(* Logix 5000 project; controller Hose_HP_Test_Rig_V1 vendor 1 type 14 code 149 rev 32.11; software revision 32.00; part 9 of 10 *)
(* tags used below, declared in another part *)
   ALIGN : SCP;
   CYCLE_TIMER_STN2 : TIMER;
   CYCLE_TIMER_STN3 : TIMER;
   GOTO_FAIL_BIN_STN1 : DINT;
   GOTO_FAULT_BIN_STN3 : DINT;
   GOTO_FAULT_BIN_STN4 : DINT;
   INDV_LTEST_ON_STN1 : BOOL;
   INDV_LTEST_ON_STN2 : BOOL;
   INDV_LTEST_ON_STN3 : BOOL;
   ONS1 : BOOL;
   ONS10 : BOOL;
   ONS11 : BOOL;
   ONS12 : BOOL;
   ONS13 : BOOL;
   ONS14 : BOOL;
   ONS15 : BOOL;
   ONS16 : BOOL;
   ONS17 : BOOL;
   ONS18 : BOOL;
   ONS19 : BOOL;
   ONS2 : BOOL;
   ONS20 : BOOL;
   ONS21 : BOOL;
   ONS22 : BOOL;
   ONS23 : BOOL;
   ONS24 : BOOL;
   ONS25 : BOOL;
   ONS3 : BOOL;
   ONS54 : BOOL;
   ONS55 : BOOL;
   ONS56 : BOOL;
   ONS57 : BOOL;
   ONS58 : BOOL;
   ONS59 : BOOL;
   ONS6 : BOOL;
   ONS60 : BOOL;
   ONS61 : BOOL;
   ONS62 : BOOL;
   ONS67 : BOOL;
   ONS68 : BOOL;
   ONS7 : BOOL;
   ONS8 : BOOL;
   ONS9 : BOOL;
   TEST_INIT_DEL_STN2 : TIMER;
   TEST_INIT_DEL_STN3 : TIMER;
   TIME1 : TIMER;
   ACT_DROP_STN1 : REAL;
   ACT_DROP_STN2 : REAL;
   ACT_DROP_STN3 : REAL;
   ACT_DROP_STN4 : REAL;
   ACT_PR_STN1 : REAL;
   ACT_PR_STN2 : REAL;
   ACT_PR_STN3 : REAL;
   ACT_PR_STN4 : REAL;
   ACT_TRAVEL : REAL;
   AUTO_DOOR_OPEN_SEQ : DINT;
   AUTO_DOOR_OPEN_SEQ_STN2 : DINT;
   AUTO_DOOR_OPEN_SEQ_STN3 : DINT;
   AUTO_TEST_ON_STN1 : BOOL;
   AUTO_TEST_ON_STN2 : BOOL;
   AUTO_TEST_ON_STN3 : BOOL;
   AUTO_TEST_ON_STN4 : BOOL;
   AUTO_TEST_OVER_STN1 : BOOL;
   AUTO_TEST_OVER_STN2 : BOOL;
   AUTO_TEST_OVER_STN3 : BOOL;
   AUTO_TEST_OVER_STN4 : BOOL;
   AUTO_TEST_SEL_STN1 : BOOL;
   AUTO_TEST_SEL_STN2 : BOOL;
   AUTO_TEST_SEL_STN3 : BOOL;
   AUTO_TEST_SEL_STN4 : BOOL;
   BOTTOM_CLAMP_PS_STN1 : ALIAS FOR Local:1:I.Data.13;
   BOTTOM_CLAMP_PS_STN2 : ALIAS FOR Local:2:I.Data.2;
   BOTTOM_CLAMP_PS_STN3 : ALIAS FOR Local:2:I.Data.7;
   BOTTOM_CLAMP_PS_STN4 : ALIAS FOR Local:2:I.Data.12;
   BOTTOM_CLAMP_SEL_STN1 : BOOL;
   BOTTOM_CLAMP_SEL_STN2 : BOOL;
   BOTTOM_CLAMP_SEL_STN3 : BOOL;
   BOTTOM_CLAMP_SEL_STN4 : BOOL;
   BOTTOM_CLAMP_SEQ_STN1 : DINT;
   BOTTOM_CLAMP_SEQ_STN2 : DINT;
   BOTTOM_CLAMP_SEQ_STN3 : DINT;
   BOTTOM_CLAMP_SET_STN1 : BOOL;
   BOTTOM_CLAMP_SET_STN2 : BOOL;
   BOTTOM_CLAMP_SET_STN3 : BOOL;
   BOTTOM_CLAMP_SET_STN4 : BOOL;
   BOTTOM_DECLAMP_SEQ_STN2 : DINT;
   BOTTOM_DECLAMP_SEQ_STN3 : DINT;
   BOTTOM_DECLAMP_SET_STN1 : BOOL;
   BOTTOM_DECLAMP_SET_STN2 : BOOL;
   BOTTOM_DECLAMP_SET_STN3 : BOOL;
   BOTTOM_DECLAMP_SET_STN4 : BOOL;
   CLR_ONS_STN1 : BOOL;
   CLR_ONS_STN2 : BOOL;
   CLR_ONS_STN3 : BOOL;
   CONS_CALB_OFF_STN1 : BOOL;
   CONS_CALB_OFF_STN2 : BOOL;
   CONS_CALB_OFF_STN3 : BOOL;
   CONS_CALB_OFF_STN4 : BOOL;
   CONS_CALB_ON_STN1 : BOOL;
   CONS_CALB_ON_STN2 : BOOL;
   CONS_CALB_ON_STN3 : BOOL;
   CONS_CALB_ON_STN4 : BOOL;
   CONS_RESULT_STN1 : DINT;
   CONS_RESULT_STN2 : DINT;
   CONS_RESULT_STN3 : DINT;
   CONS_RESULT_STN4 : DINT;
   CONS_STS_STN1 : DINT;
   CONS_STS_STN2 : DINT;
   CONS_STS_STN3 : DINT;
   CONS_STS_STN4 : DINT;
   CONS_TEST_ON : BOOL;
   CONSTRICTION_CALB_SEL_STN1 : BOOL;
   CONSTRICTION_CALB_SEL_STN2 : BOOL;
   CONSTRICTION_CALB_SEL_STN3 : BOOL;
   CONSTRICTION_CALB_SEL_STN4 : BOOL;
   CONSTRICTION_VALVE_STN1 : BOOL;
   CONSTRICTION_VALVE_STN2 : BOOL;
   CONSTRICTION_VALVE_STN3 : BOOL;
   CONSTRICTION_VALVE_STN4 : BOOL;
   CRIMP_PASS : ALIAS FOR Local:2:I.Data.31;
   CRIMP_PASS_TO_TRACE : DINT;
   CYCLE_START_PB_STN1 : ALIAS FOR Local:1:I.Data.2;
   CYCLE_TIME_ACT_STN1 : REAL;
   CYCLE_TIME_ACT_STN2 : REAL;
   CYCLE_TIME_ACT_STN3 : REAL;
   CYCLE_TIME_ACT_STN4 : REAL;
   CYCLE_TIMER_STN1 : TIMER;
   CYCLE_TIMER_STN4 : TIMER;
   DOOR_CLAMP_SET_STN1 : SETTING_MODE;
   DOOR_CLAMP_SET_STN2 : SETTING_MODE;
   DOOR_CLAMP_SET_STN3 : SETTING_MODE;
   DOOR_CLAMP_SET_STN4 : SETTING_MODE;
   DOOR_CLOSE_SEL_STN1 : BOOL;
   DOOR_CLOSE_SEL_STN2 : BOOL;
   DOOR_CLOSE_SEL_STN3 : BOOL;
   DOOR_CLOSE_SEL_STN4 : BOOL;
   DOOR_CLOSE_SET_STN1 : BOOL;
   DOOR_CLOSE_SET_STN2 : BOOL;
   DOOR_CLOSE_SET_STN3 : BOOL;
   DOOR_CLOSE_SET_STN4 : BOOL;
   DOOR_OPEN_RS_STN1 : ALIAS FOR Local:1:I.Data.10;
   DOOR_OPEN_RS_STN2 : ALIAS FOR Local:1:I.Data.15;
   DOOR_OPEN_RS_STN3 : ALIAS FOR Local:2:I.Data.4;
   DOOR_OPEN_RS_STN4 : ALIAS FOR Local:2:I.Data.10;
   DOOR_OPEN_SET_STN1 : BOOL;
   DOOR_OPEN_SET_STN2 : BOOL;
   DOOR_OPEN_SET_STN3 : BOOL;
   DOOR_OPEN_SET_STN4 : BOOL;
   EXHAUST_SET_STN1 : BOOL;
   EXHAUST_SET_STN2 : BOOL;
   EXHAUST_SET_STN3 : BOOL;
   EXHAUST_SET_STN4 : BOOL;
   EXHAUST_VALVE_STN1 : ALIAS FOR Local:1:O.Data.7;
   EXHAUST_VALVE_STN2 : ALIAS FOR Local:1:O.Data.15;
   EXHAUST_VALVE_STN3 : ALIAS FOR Local:3:O.Data.7;
   EXHAUST_VALVE_STN4 : ALIAS FOR Local:3:O.Data.15;
   FAIL_BIN_DOOR_PROXY : ALIAS FOR Local:2:I.Data.29;
   FAILED_STN1 : BOOL;
   FAILED_STN2 : BOOL;
   FAILED_STN3 : BOOL;
   FAILED_STN4 : BOOL;
   FAULTED_STN1 : BOOL;
   FAULTED_STN2 : BOOL;
   FAULTED_STN3 : BOOL;
   FAULTED_STN4 : BOOL;
   FIX_DOWN_SET : BOOL;
   FIX_UP_SET : BOOL;
   GOTO_FAIL_BIN_STN2 : DINT;
   GOTO_FAIL_BIN_STN3 : DINT;
   GOTO_FAIL_BIN_STN4 : DINT;
   GOTO_FAULT_BIN_STN1 : DINT;
   GOTO_FAULT_BIN_STN2 : DINT;
   HOME_COND_OK_STN1 : BOOL;
   HOME_COND_OK_STN2 : BOOL;
   HOME_COND_OK_STN3 : BOOL;
   HOME_COND_OK_STN4 : BOOL;
   HP_ACT_DROP_STN1 : REAL;
   HP_ACT_DROP_STN2 : REAL;
   HP_ACT_DROP_STN3 : REAL;
   HP_ACT_DROP_STN4 : REAL;
   HP_ACT_PR_STN1 : REAL;
   HP_ACT_PR_STN2 : REAL;
   HP_ACT_PR_STN3 : REAL;
   HP_ACT_PR_STN4 : REAL;
   HP_RESULT_STN1 : DINT;
   HP_RESULT_STN2 : DINT;
   HP_RESULT_STN3 : DINT;
   HP_RESULT_STN4 : DINT;
   HP_SENSOR_SEL : BOOL;
   HP_STS_STN1 : DINT;
   HP_STS_STN2 : DINT;
   HP_STS_STN3 : DINT;
   HP_STS_STN4 : DINT;
   HP_TEST_ON : BOOL;
   INDV_CTEST_ON_STN1 : BOOL;
   INDV_CTEST_ON_STN2 : BOOL;
   INDV_CTEST_ON_STN3 : BOOL;
   INIT_STN1 : BOOL;
   INIT_STN2 : BOOL;
   INIT_STN3 : BOOL;
   LH_START_PB_STN2 : ALIAS FOR Local:1:I.Data.3;
   LH_START_PB_STN3 : ALIAS FOR Local:1:I.Data.4;
   LH_START_PB_STN4 : ALIAS FOR Local:1:I.Data.5;
   LOGIN_LEVEL : INT;
   MASTER_WORK_MAIN_MENU_EN : BOOL;
   MOTOR_DOWN : ALIAS FOR REM:O.Data[1].3;
   MOTOR_SAFETY : BOOL;
   MOTOR_UP : ALIAS FOR REM:O.Data[1].2;
   MSG_STN1 : DINT;
   MSG_STN2 : DINT;
   MSG_STN3 : DINT;
   MSG_STN4 : DINT;
   ONS5 : BOOL;
   OTHER_CAL_EDIT_MODE : BOOL;
   OTHER_CAL_VIEW_MODE : BOOL;
   OTHER_SENSOR_SEL : BOOL;
   PASSED_STN1 : BOOL;
   PASSED_STN2 : BOOL;
   PASSED_STN3 : BOOL;
   RETEST : BOOL;
   RST_SEQ_ON_STN1 : BOOL;
   RST_SEQ_ON_STN2 : BOOL;
   RST_SEQ_ON_STN3 : BOOL;
   RST_SEQ_ON_STN4 : BOOL;
   SCR_STS : DINT[6];
   SENS_CAL_EDIT_MODE : BOOL;
   SENS_CAL_SEL_BOTTOM_CLAMP : BOOL;
   SENS_CAL_SEL_MASTER : BOOL;
   SENS_CAL_SEL_STAMP : BOOL;
   SENS_CAL_SEL_TOP_CLAMP : BOOL;
   SENS_CAL_VIEW_MODE : BOOL;
   SENS_CALB_SEL_STN1 : BOOL;
   SENS_CALB_SEL_STN2 : BOOL;
   SENS_CALB_SEL_STN3 : BOOL;
   SENS_CALB_SEL_STN4 : BOOL;
   SEQ_NO_STN1 : DINT;
   SEQ_NO_STN2 : DINT;
   SEQ_NO_STN3 : DINT;
   SET_240 : REAL;
   SET_DISTANCE : REAL;
   SET_MENU_STN1_EN : BOOL;
   SET_MENU_STN2_EN : BOOL;
   SET_MENU_STN3_EN : BOOL;
   SET_MENU_STN4_EN : BOOL;
   SET_MODE_SEL_STN1 : BOOL;
   SET_MODE_SEL_STN2 : BOOL;
   SET_MODE_SEL_STN3 : BOOL;
   SET_MODE_SEL_STN4 : BOOL;
   SET_TIMER : REAL;
   SLIDE_TRAVEL : TIMER;
(* MainProgram, continued *)

ROUTINE SENS_CALB   (* ladder *)
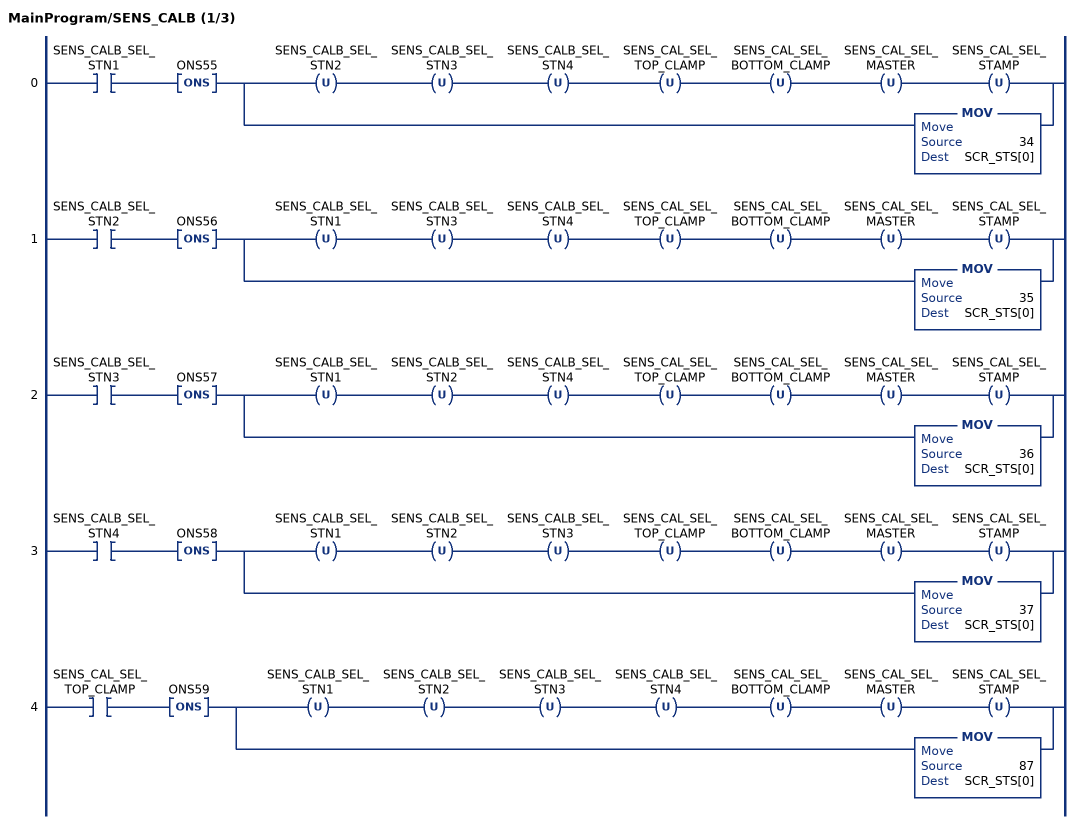
   0: XIC(SENS_CALB_SEL_STN1)ONS(ONS55)[OTU(SENS_CALB_SEL_STN2) OTU(SENS_CALB_SEL_STN3) OTU(SENS_CALB_SEL_STN4) OTU(SENS_CAL_SEL_TOP_CLAMP) OTU(SENS_CAL_SEL_BOTTOM_CLAMP) OTU(SENS_CAL_SEL_MASTER) OTU(SENS_CAL_SEL_STAMP) ,MOV(34,SCR_STS[0]) ];
   1: XIC(SENS_CALB_SEL_STN2)ONS(ONS56)[OTU(SENS_CALB_SEL_STN1) OTU(SENS_CALB_SEL_STN3) OTU(SENS_CALB_SEL_STN4) OTU(SENS_CAL_SEL_TOP_CLAMP) OTU(SENS_CAL_SEL_BOTTOM_CLAMP) OTU(SENS_CAL_SEL_MASTER) OTU(SENS_CAL_SEL_STAMP) ,MOV(35,SCR_STS[0]) ];
   2: XIC(SENS_CALB_SEL_STN3)ONS(ONS57)[OTU(SENS_CALB_SEL_STN1) OTU(SENS_CALB_SEL_STN2) OTU(SENS_CALB_SEL_STN4) OTU(SENS_CAL_SEL_TOP_CLAMP) OTU(SENS_CAL_SEL_BOTTOM_CLAMP) OTU(SENS_CAL_SEL_MASTER) OTU(SENS_CAL_SEL_STAMP) ,MOV(36,SCR_STS[0]) ];
   3: XIC(SENS_CALB_SEL_STN4)ONS(ONS58)[OTU(SENS_CALB_SEL_STN1) OTU(SENS_CALB_SEL_STN2) OTU(SENS_CALB_SEL_STN3) OTU(SENS_CAL_SEL_TOP_CLAMP) OTU(SENS_CAL_SEL_BOTTOM_CLAMP) OTU(SENS_CAL_SEL_MASTER) OTU(SENS_CAL_SEL_STAMP) ,MOV(37,SCR_STS[0]) ];
   4: XIC(SENS_CAL_SEL_TOP_CLAMP)ONS(ONS59)[OTU(SENS_CALB_SEL_STN1) OTU(SENS_CALB_SEL_STN2) OTU(SENS_CALB_SEL_STN3) OTU(SENS_CALB_SEL_STN4) OTU(SENS_CAL_SEL_BOTTOM_CLAMP) OTU(SENS_CAL_SEL_MASTER) OTU(SENS_CAL_SEL_STAMP) ,MOV(87,SCR_STS[0]) ];
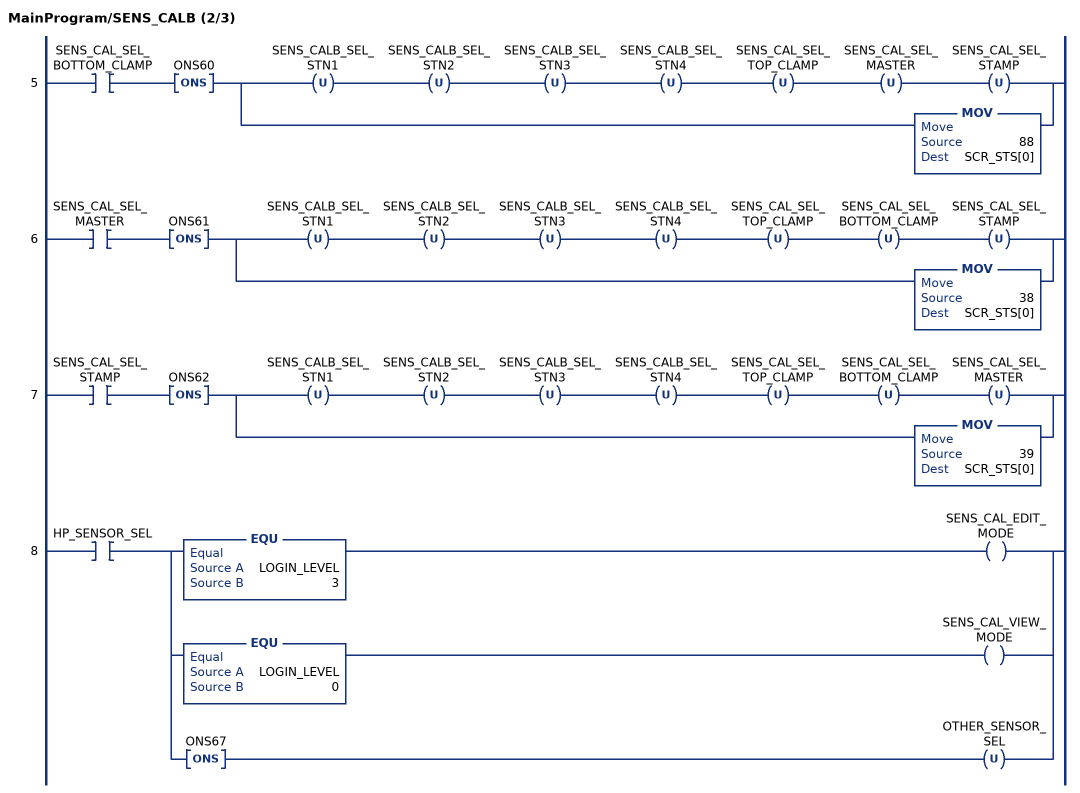
   5: XIC(SENS_CAL_SEL_BOTTOM_CLAMP)ONS(ONS60)[OTU(SENS_CALB_SEL_STN1) OTU(SENS_CALB_SEL_STN2) OTU(SENS_CALB_SEL_STN3) OTU(SENS_CALB_SEL_STN4) OTU(SENS_CAL_SEL_TOP_CLAMP) OTU(SENS_CAL_SEL_MASTER) OTU(SENS_CAL_SEL_STAMP) ,MOV(88,SCR_STS[0]) ];
   6: XIC(SENS_CAL_SEL_MASTER)ONS(ONS61)[OTU(SENS_CALB_SEL_STN1) OTU(SENS_CALB_SEL_STN2) OTU(SENS_CALB_SEL_STN3) OTU(SENS_CALB_SEL_STN4) OTU(SENS_CAL_SEL_TOP_CLAMP) OTU(SENS_CAL_SEL_BOTTOM_CLAMP) OTU(SENS_CAL_SEL_STAMP) ,MOV(38,SCR_STS[0]) ];
   7: XIC(SENS_CAL_SEL_STAMP)ONS(ONS62)[OTU(SENS_CALB_SEL_STN1) OTU(SENS_CALB_SEL_STN2) OTU(SENS_CALB_SEL_STN3) OTU(SENS_CALB_SEL_STN4) OTU(SENS_CAL_SEL_TOP_CLAMP) OTU(SENS_CAL_SEL_BOTTOM_CLAMP) OTU(SENS_CAL_SEL_MASTER) ,MOV(39,SCR_STS[0]) ];
   8: XIC(HP_SENSOR_SEL)[EQU(LOGIN_LEVEL,3) OTE(SENS_CAL_EDIT_MODE) ,EQU(LOGIN_LEVEL,0) OTE(SENS_CAL_VIEW_MODE) ,ONS(ONS67) OTU(OTHER_SENSOR_SEL) ];
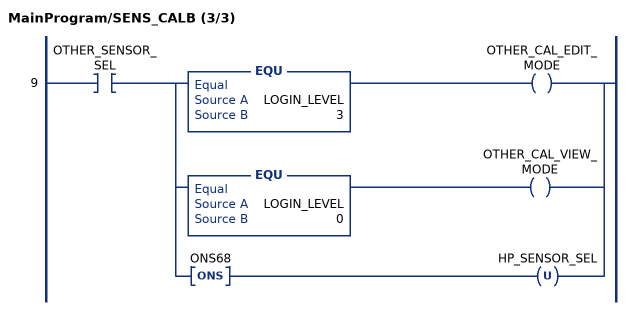
   9: XIC(OTHER_SENSOR_SEL)[EQU(LOGIN_LEVEL,3) OTE(OTHER_CAL_EDIT_MODE) ,EQU(LOGIN_LEVEL,0) OTE(OTHER_CAL_VIEW_MODE) ,ONS(ONS68) OTU(HP_SENSOR_SEL) ];
END_ROUTINE

ROUTINE Setting_Mode   (* ladder *)
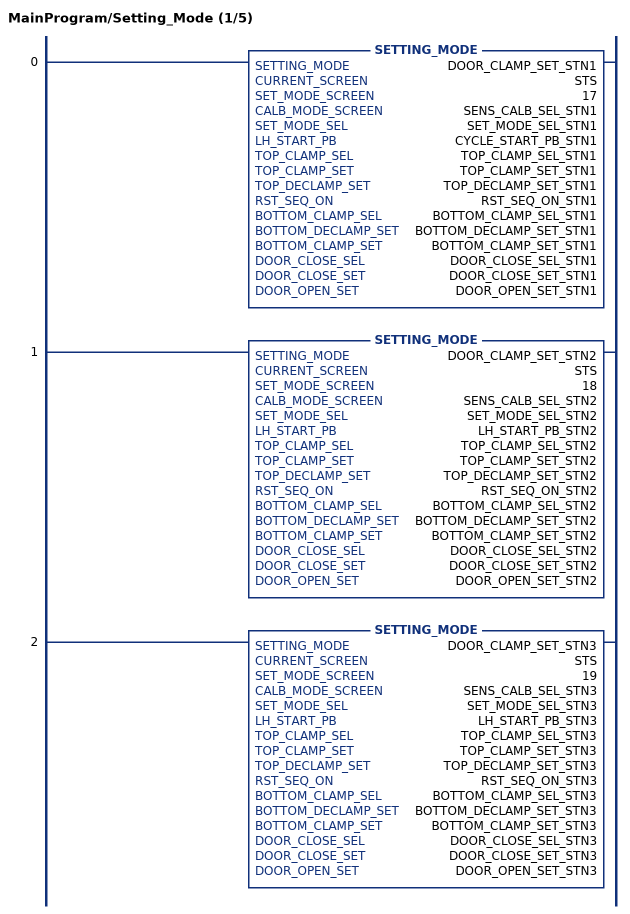
   0: SETTING_MODE(DOOR_CLAMP_SET_STN1,STS,17,SENS_CALB_SEL_STN1,SET_MODE_SEL_STN1,CYCLE_START_PB_STN1,TOP_CLAMP_SEL_STN1,TOP_CLAMP_SET_STN1,TOP_DECLAMP_SET_STN1,RST_SEQ_ON_STN1,BOTTOM_CLAMP_SEL_STN1,BOTTOM_DECLAMP_SET_STN1,BOTTOM_CLAMP_SET_STN1,DOOR_CLOSE_SEL_STN1,DOOR_CLOSE_SET_STN1,DOOR_OPEN_SET_STN1);
   1: SETTING_MODE(DOOR_CLAMP_SET_STN2,STS,18,SENS_CALB_SEL_STN2,SET_MODE_SEL_STN2,LH_START_PB_STN2,TOP_CLAMP_SEL_STN2,TOP_CLAMP_SET_STN2,TOP_DECLAMP_SET_STN2,RST_SEQ_ON_STN2,BOTTOM_CLAMP_SEL_STN2,BOTTOM_DECLAMP_SET_STN2,BOTTOM_CLAMP_SET_STN2,DOOR_CLOSE_SEL_STN2,DOOR_CLOSE_SET_STN2,DOOR_OPEN_SET_STN2);
   2: SETTING_MODE(DOOR_CLAMP_SET_STN3,STS,19,SENS_CALB_SEL_STN3,SET_MODE_SEL_STN3,LH_START_PB_STN3,TOP_CLAMP_SEL_STN3,TOP_CLAMP_SET_STN3,TOP_DECLAMP_SET_STN3,RST_SEQ_ON_STN3,BOTTOM_CLAMP_SEL_STN3,BOTTOM_DECLAMP_SET_STN3,BOTTOM_CLAMP_SET_STN3,DOOR_CLOSE_SEL_STN3,DOOR_CLOSE_SET_STN3,DOOR_OPEN_SET_STN3);
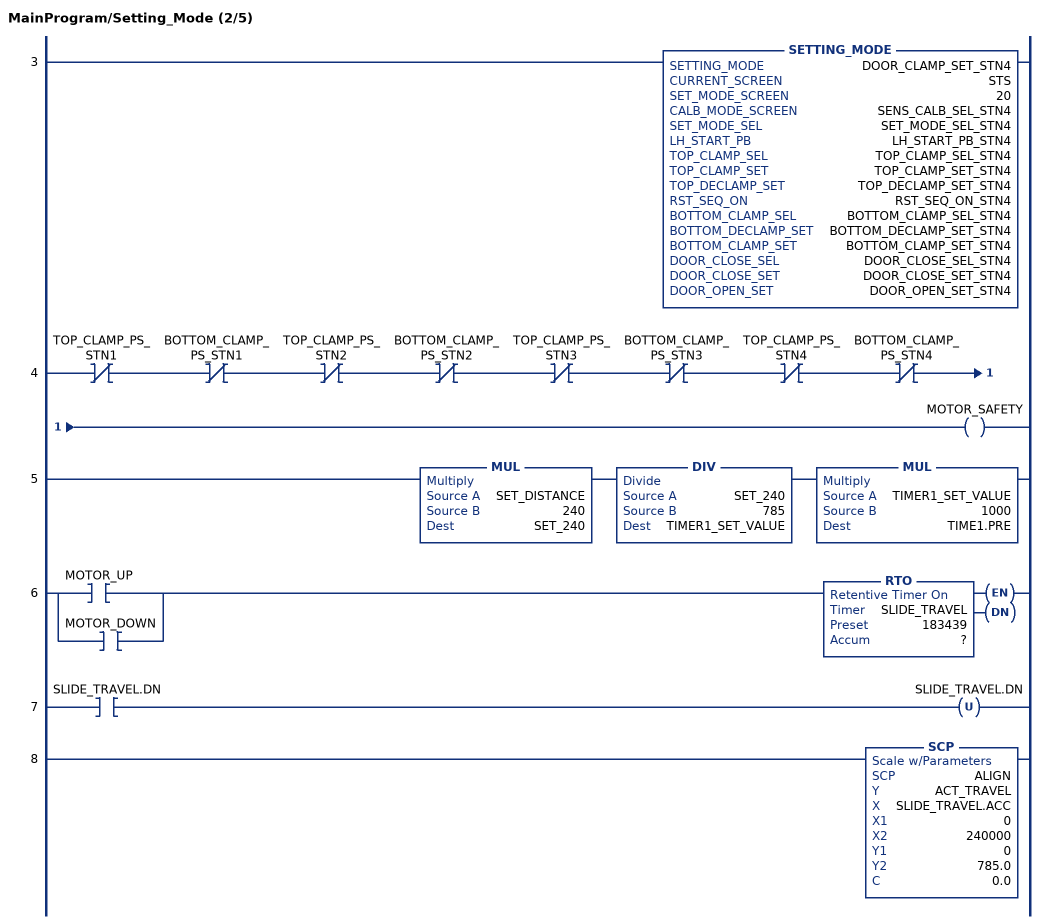
   3: SETTING_MODE(DOOR_CLAMP_SET_STN4,STS,20,SENS_CALB_SEL_STN4,SET_MODE_SEL_STN4,LH_START_PB_STN4,TOP_CLAMP_SEL_STN4,TOP_CLAMP_SET_STN4,TOP_DECLAMP_SET_STN4,RST_SEQ_ON_STN4,BOTTOM_CLAMP_SEL_STN4,BOTTOM_DECLAMP_SET_STN4,BOTTOM_CLAMP_SET_STN4,DOOR_CLOSE_SEL_STN4,DOOR_CLOSE_SET_STN4,DOOR_OPEN_SET_STN4);
   4: XIO(TOP_CLAMP_PS_STN1)XIO(BOTTOM_CLAMP_PS_STN1)XIO(TOP_CLAMP_PS_STN2)XIO(BOTTOM_CLAMP_PS_STN2)XIO(TOP_CLAMP_PS_STN3)XIO(BOTTOM_CLAMP_PS_STN3)XIO(TOP_CLAMP_PS_STN4)XIO(BOTTOM_CLAMP_PS_STN4)OTE(MOTOR_SAFETY);
   5: MUL(SET_DISTANCE,240,SET_240)DIV(SET_240,785,TIMER1_SET_VALUE)MUL(TIMER1_SET_VALUE,1000,TIME1.PRE);
   6: [XIC(MOTOR_UP) ,XIC(MOTOR_DOWN) ]RTO(SLIDE_TRAVEL,?,?);
   7: XIC(SLIDE_TRAVEL.DN)OTU(SLIDE_TRAVEL.DN);
   8: SCP(ALIGN,ACT_TRAVEL,SLIDE_TRAVEL.ACC,0,240000,0,785.0,0.0);
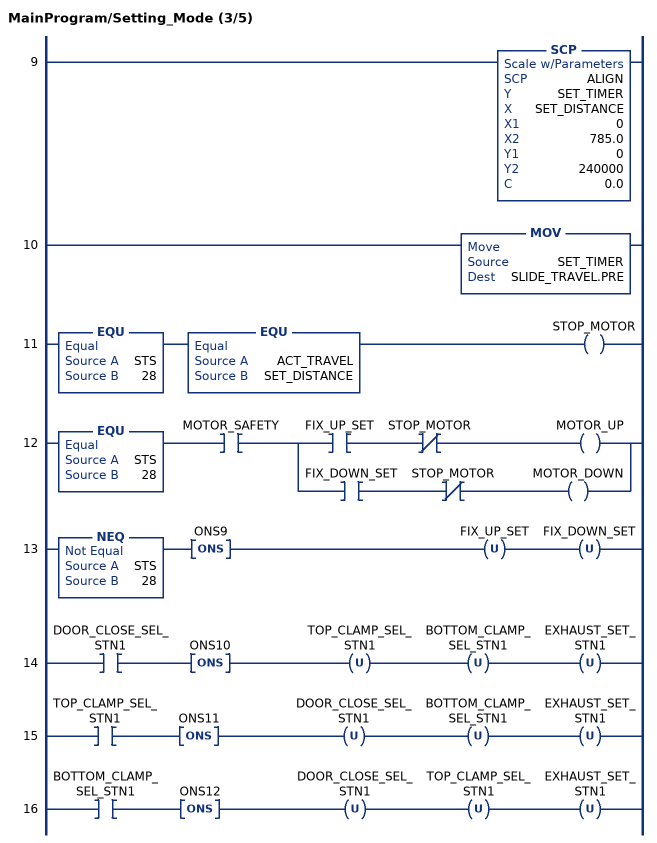
   9: SCP(ALIGN,SET_TIMER,SET_DISTANCE,0,785.0,0,240000,0.0);
   10: MOV(SET_TIMER,SLIDE_TRAVEL.PRE);
   11: EQU(STS,28)EQU(ACT_TRAVEL,SET_DISTANCE)OTE(STOP_MOTOR);
   12: EQU(STS,28)XIC(MOTOR_SAFETY)[XIC(FIX_UP_SET) XIO(STOP_MOTOR) OTE(MOTOR_UP) ,XIC(FIX_DOWN_SET) XIO(STOP_MOTOR) OTE(MOTOR_DOWN) ];
   13: NEQ(STS,28)ONS(ONS9)OTU(FIX_UP_SET)OTU(FIX_DOWN_SET);
   14: XIC(DOOR_CLOSE_SEL_STN1)ONS(ONS10)OTU(TOP_CLAMP_SEL_STN1)OTU(BOTTOM_CLAMP_SEL_STN1)OTU(EXHAUST_SET_STN1);
   15: XIC(TOP_CLAMP_SEL_STN1)ONS(ONS11)OTU(DOOR_CLOSE_SEL_STN1)OTU(BOTTOM_CLAMP_SEL_STN1)OTU(EXHAUST_SET_STN1);
   16: XIC(BOTTOM_CLAMP_SEL_STN1)ONS(ONS12)OTU(DOOR_CLOSE_SEL_STN1)OTU(TOP_CLAMP_SEL_STN1)OTU(EXHAUST_SET_STN1);
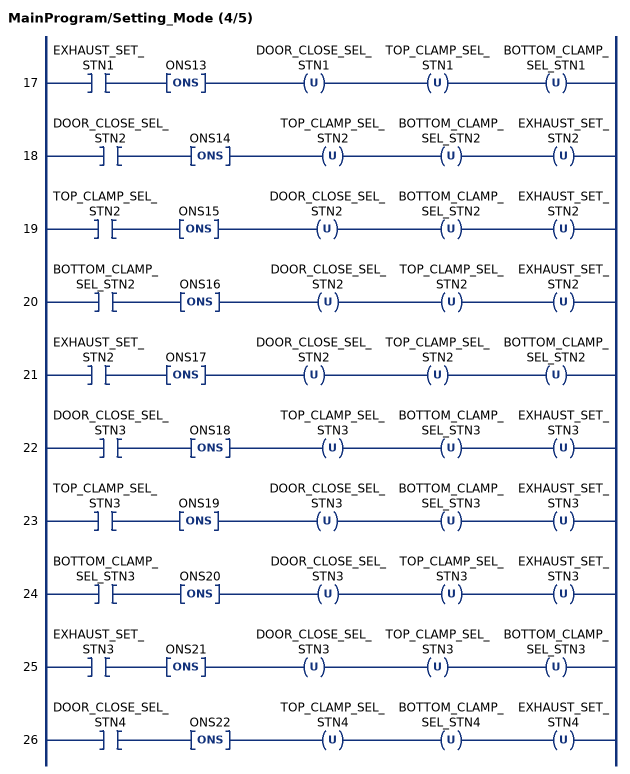
   17: XIC(EXHAUST_SET_STN1)ONS(ONS13)OTU(DOOR_CLOSE_SEL_STN1)OTU(TOP_CLAMP_SEL_STN1)OTU(BOTTOM_CLAMP_SEL_STN1);
   18: XIC(DOOR_CLOSE_SEL_STN2)ONS(ONS14)OTU(TOP_CLAMP_SEL_STN2)OTU(BOTTOM_CLAMP_SEL_STN2)OTU(EXHAUST_SET_STN2);
   19: XIC(TOP_CLAMP_SEL_STN2)ONS(ONS15)OTU(DOOR_CLOSE_SEL_STN2)OTU(BOTTOM_CLAMP_SEL_STN2)OTU(EXHAUST_SET_STN2);
   20: XIC(BOTTOM_CLAMP_SEL_STN2)ONS(ONS16)OTU(DOOR_CLOSE_SEL_STN2)OTU(TOP_CLAMP_SEL_STN2)OTU(EXHAUST_SET_STN2);
   21: XIC(EXHAUST_SET_STN2)ONS(ONS17)OTU(DOOR_CLOSE_SEL_STN2)OTU(TOP_CLAMP_SEL_STN2)OTU(BOTTOM_CLAMP_SEL_STN2);
   22: XIC(DOOR_CLOSE_SEL_STN3)ONS(ONS18)OTU(TOP_CLAMP_SEL_STN3)OTU(BOTTOM_CLAMP_SEL_STN3)OTU(EXHAUST_SET_STN3);
   23: XIC(TOP_CLAMP_SEL_STN3)ONS(ONS19)OTU(DOOR_CLOSE_SEL_STN3)OTU(BOTTOM_CLAMP_SEL_STN3)OTU(EXHAUST_SET_STN3);
   24: XIC(BOTTOM_CLAMP_SEL_STN3)ONS(ONS20)OTU(DOOR_CLOSE_SEL_STN3)OTU(TOP_CLAMP_SEL_STN3)OTU(EXHAUST_SET_STN3);
   25: XIC(EXHAUST_SET_STN3)ONS(ONS21)OTU(DOOR_CLOSE_SEL_STN3)OTU(TOP_CLAMP_SEL_STN3)OTU(BOTTOM_CLAMP_SEL_STN3);
   26: XIC(DOOR_CLOSE_SEL_STN4)ONS(ONS22)OTU(TOP_CLAMP_SEL_STN4)OTU(BOTTOM_CLAMP_SEL_STN4)OTU(EXHAUST_SET_STN4);
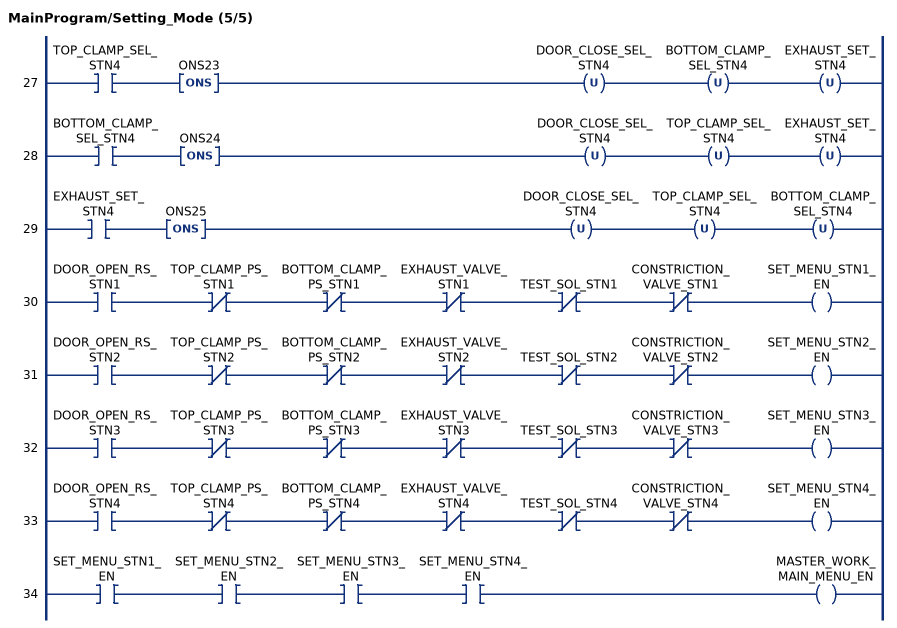
   27: XIC(TOP_CLAMP_SEL_STN4)ONS(ONS23)OTU(DOOR_CLOSE_SEL_STN4)OTU(BOTTOM_CLAMP_SEL_STN4)OTU(EXHAUST_SET_STN4);
   28: XIC(BOTTOM_CLAMP_SEL_STN4)ONS(ONS24)OTU(DOOR_CLOSE_SEL_STN4)OTU(TOP_CLAMP_SEL_STN4)OTU(EXHAUST_SET_STN4);
   29: XIC(EXHAUST_SET_STN4)ONS(ONS25)OTU(DOOR_CLOSE_SEL_STN4)OTU(TOP_CLAMP_SEL_STN4)OTU(BOTTOM_CLAMP_SEL_STN4);
   30: XIC(DOOR_OPEN_RS_STN1)XIO(TOP_CLAMP_PS_STN1)XIO(BOTTOM_CLAMP_PS_STN1)XIO(EXHAUST_VALVE_STN1)XIO(TEST_SOL_STN1)XIO(CONSTRICTION_VALVE_STN1)OTE(SET_MENU_STN1_EN);
   31: XIC(DOOR_OPEN_RS_STN2)XIO(TOP_CLAMP_PS_STN2)XIO(BOTTOM_CLAMP_PS_STN2)XIO(EXHAUST_VALVE_STN2)XIO(TEST_SOL_STN2)XIO(CONSTRICTION_VALVE_STN2)OTE(SET_MENU_STN2_EN);
   32: XIC(DOOR_OPEN_RS_STN3)XIO(TOP_CLAMP_PS_STN3)XIO(BOTTOM_CLAMP_PS_STN3)XIO(EXHAUST_VALVE_STN3)XIO(TEST_SOL_STN3)XIO(CONSTRICTION_VALVE_STN3)OTE(SET_MENU_STN3_EN);
   33: XIC(DOOR_OPEN_RS_STN4)XIO(TOP_CLAMP_PS_STN4)XIO(BOTTOM_CLAMP_PS_STN4)XIO(EXHAUST_VALVE_STN4)XIO(TEST_SOL_STN4)XIO(CONSTRICTION_VALVE_STN4)OTE(SET_MENU_STN4_EN);
   34: XIC(SET_MENU_STN1_EN)XIC(SET_MENU_STN2_EN)XIC(SET_MENU_STN3_EN)XIC(SET_MENU_STN4_EN)OTE(MASTER_WORK_MAIN_MENU_EN);
END_ROUTINE

ROUTINE TRACEABILITY   (* ladder *)
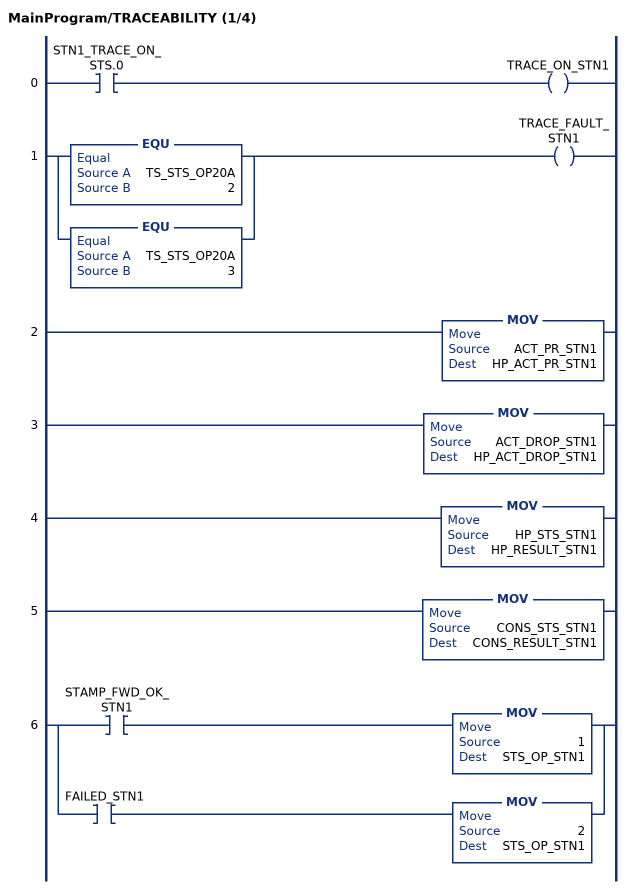
   0: XIC(STN1_TRACE_ON_STS.0)OTE(TRACE_ON_STN1);
   1: [EQU(TS_STS_OP20A,2) ,EQU(TS_STS_OP20A,3) ]OTE(TRACE_FAULT_STN1);
   2: MOV(ACT_PR_STN1,HP_ACT_PR_STN1);
   3: MOV(ACT_DROP_STN1,HP_ACT_DROP_STN1);
   4: MOV(HP_STS_STN1,HP_RESULT_STN1);
   5: MOV(CONS_STS_STN1,CONS_RESULT_STN1);
   6: [XIC(STAMP_FWD_OK_STN1) MOV(1,STS_OP_STN1) ,XIC(FAILED_STN1) MOV(2,STS_OP_STN1) ];
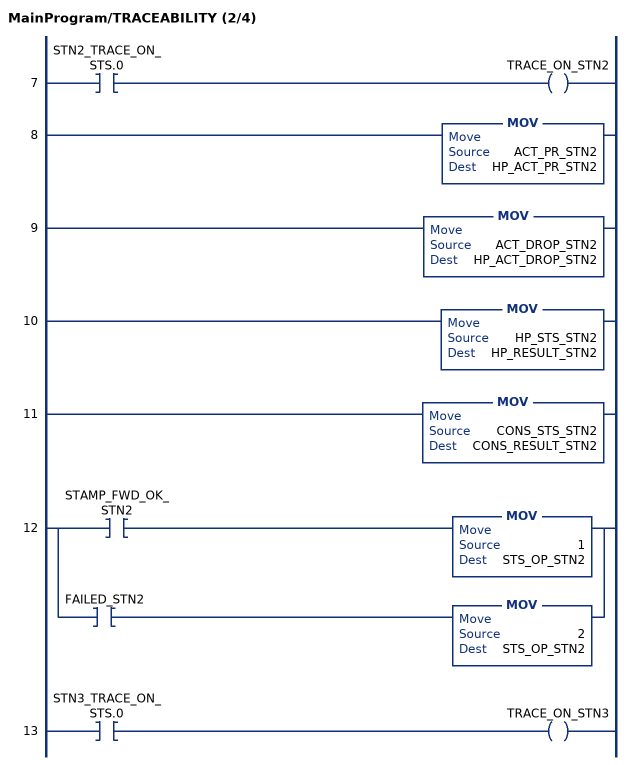
   7: XIC(STN2_TRACE_ON_STS.0)OTE(TRACE_ON_STN2);
   8: MOV(ACT_PR_STN2,HP_ACT_PR_STN2);
   9: MOV(ACT_DROP_STN2,HP_ACT_DROP_STN2);
   10: MOV(HP_STS_STN2,HP_RESULT_STN2);
   11: MOV(CONS_STS_STN2,CONS_RESULT_STN2);
   12: [XIC(STAMP_FWD_OK_STN2) MOV(1,STS_OP_STN2) ,XIC(FAILED_STN2) MOV(2,STS_OP_STN2) ];
   13: XIC(STN3_TRACE_ON_STS.0)OTE(TRACE_ON_STN3);
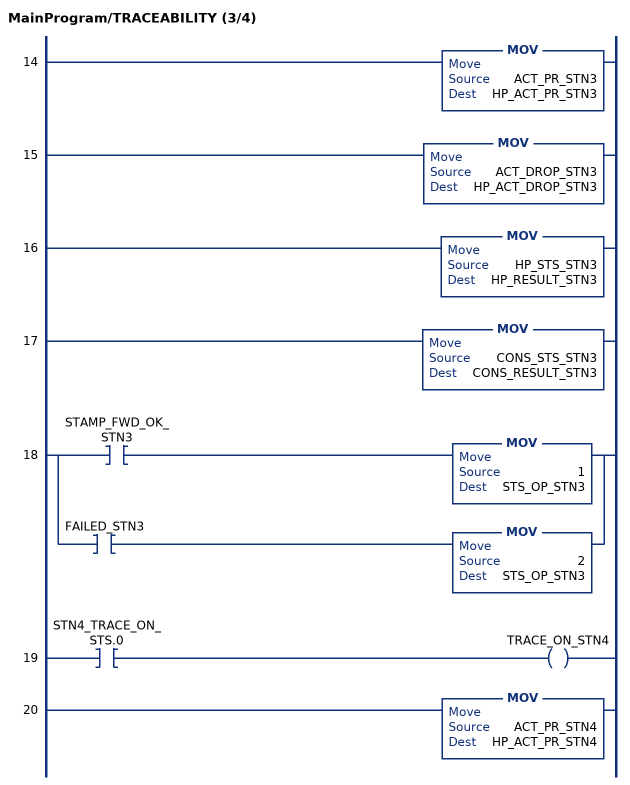
   14: MOV(ACT_PR_STN3,HP_ACT_PR_STN3);
   15: MOV(ACT_DROP_STN3,HP_ACT_DROP_STN3);
   16: MOV(HP_STS_STN3,HP_RESULT_STN3);
   17: MOV(CONS_STS_STN3,CONS_RESULT_STN3);
   18: [XIC(STAMP_FWD_OK_STN3) MOV(1,STS_OP_STN3) ,XIC(FAILED_STN3) MOV(2,STS_OP_STN3) ];
   19: XIC(STN4_TRACE_ON_STS.0)OTE(TRACE_ON_STN4);
   20: MOV(ACT_PR_STN4,HP_ACT_PR_STN4);
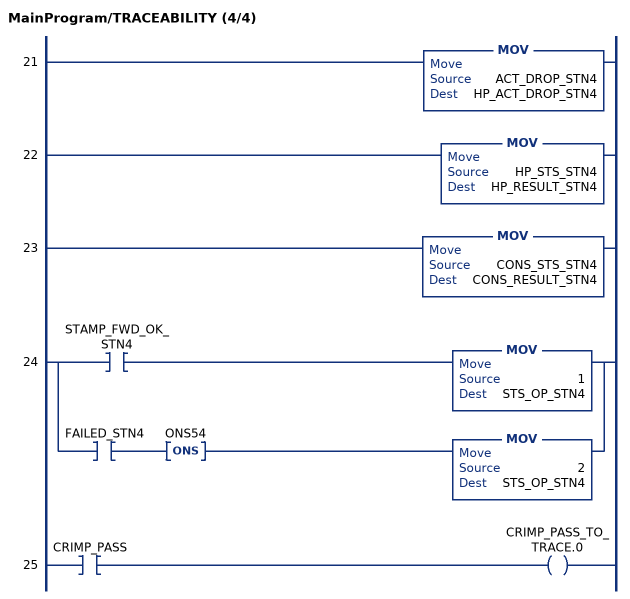
   21: MOV(ACT_DROP_STN4,HP_ACT_DROP_STN4);
   22: MOV(HP_STS_STN4,HP_RESULT_STN4);
   23: MOV(CONS_STS_STN4,CONS_RESULT_STN4);
   24: [XIC(STAMP_FWD_OK_STN4) MOV(1,STS_OP_STN4) ,XIC(FAILED_STN4) ONS(ONS54) MOV(2,STS_OP_STN4) ];
   25: XIC(CRIMP_PASS)OTE(CRIMP_PASS_TO_TRACE.0);
END_ROUTINE

ROUTINE Which_Scr_Test   (* ladder *)
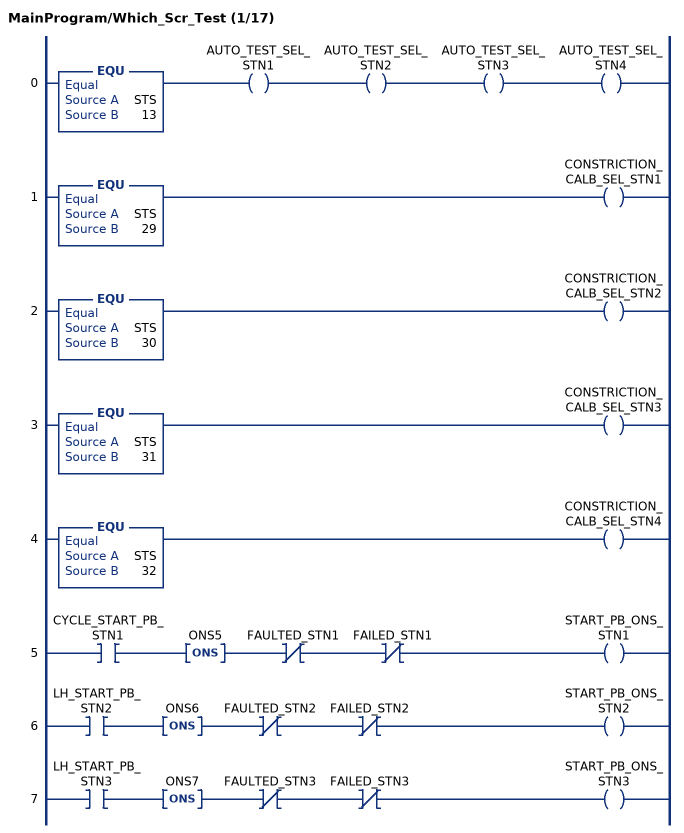
   0: EQU(STS,13)OTE(AUTO_TEST_SEL_STN1)OTE(AUTO_TEST_SEL_STN2)OTE(AUTO_TEST_SEL_STN3)OTE(AUTO_TEST_SEL_STN4);
   1: EQU(STS,29)OTE(CONSTRICTION_CALB_SEL_STN1);
   2: EQU(STS,30)OTE(CONSTRICTION_CALB_SEL_STN2);
   3: EQU(STS,31)OTE(CONSTRICTION_CALB_SEL_STN3);
   4: EQU(STS,32)OTE(CONSTRICTION_CALB_SEL_STN4);
   5: XIC(CYCLE_START_PB_STN1)ONS(ONS5)XIO(FAULTED_STN1)XIO(FAILED_STN1)OTE(START_PB_ONS_STN1);
   6: XIC(LH_START_PB_STN2)ONS(ONS6)XIO(FAULTED_STN2)XIO(FAILED_STN2)OTE(START_PB_ONS_STN2);
   7: XIC(LH_START_PB_STN3)ONS(ONS7)XIO(FAULTED_STN3)XIO(FAILED_STN3)OTE(START_PB_ONS_STN3);
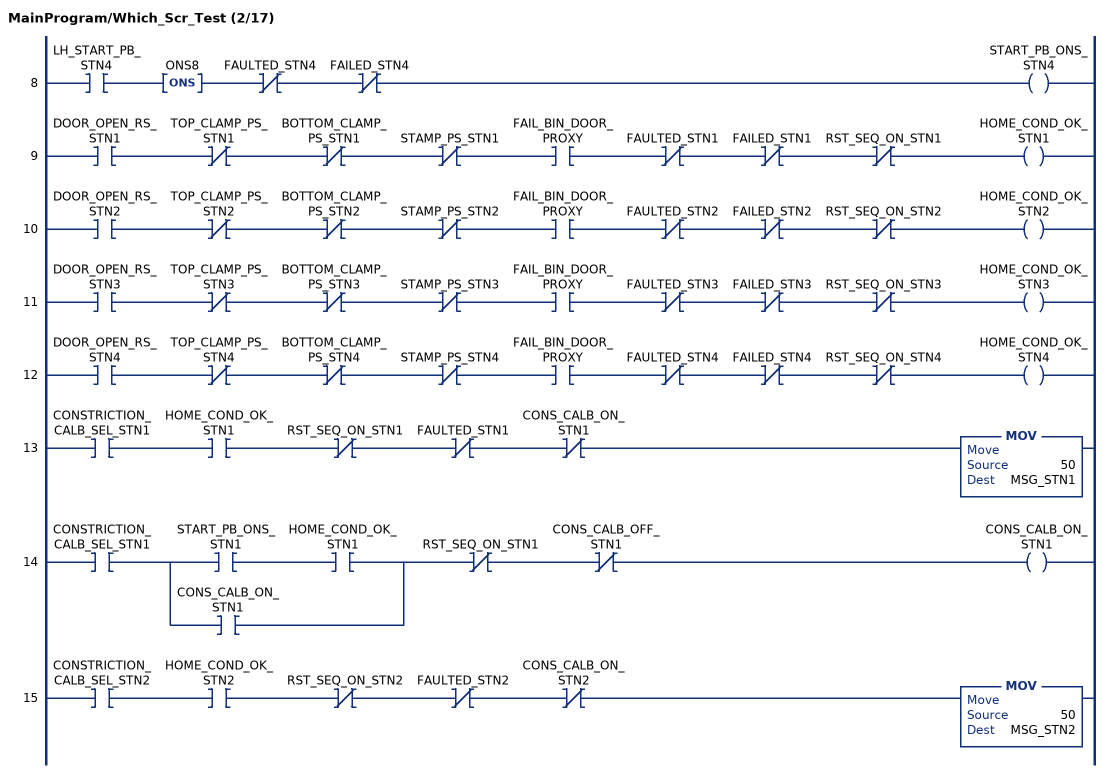
   8: XIC(LH_START_PB_STN4)ONS(ONS8)XIO(FAULTED_STN4)XIO(FAILED_STN4)OTE(START_PB_ONS_STN4);
   9: XIC(DOOR_OPEN_RS_STN1)XIO(TOP_CLAMP_PS_STN1)XIO(BOTTOM_CLAMP_PS_STN1)XIO(STAMP_PS_STN1)XIC(FAIL_BIN_DOOR_PROXY)XIO(FAULTED_STN1)XIO(FAILED_STN1)XIO(RST_SEQ_ON_STN1)OTE(HOME_COND_OK_STN1);
   10: XIC(DOOR_OPEN_RS_STN2)XIO(TOP_CLAMP_PS_STN2)XIO(BOTTOM_CLAMP_PS_STN2)XIO(STAMP_PS_STN2)XIC(FAIL_BIN_DOOR_PROXY)XIO(FAULTED_STN2)XIO(FAILED_STN2)XIO(RST_SEQ_ON_STN2)OTE(HOME_COND_OK_STN2);
   11: XIC(DOOR_OPEN_RS_STN3)XIO(TOP_CLAMP_PS_STN3)XIO(BOTTOM_CLAMP_PS_STN3)XIO(STAMP_PS_STN3)XIC(FAIL_BIN_DOOR_PROXY)XIO(FAULTED_STN3)XIO(FAILED_STN3)XIO(RST_SEQ_ON_STN3)OTE(HOME_COND_OK_STN3);
   12: XIC(DOOR_OPEN_RS_STN4)XIO(TOP_CLAMP_PS_STN4)XIO(BOTTOM_CLAMP_PS_STN4)XIO(STAMP_PS_STN4)XIC(FAIL_BIN_DOOR_PROXY)XIO(FAULTED_STN4)XIO(FAILED_STN4)XIO(RST_SEQ_ON_STN4)OTE(HOME_COND_OK_STN4);
   13: XIC(CONSTRICTION_CALB_SEL_STN1)XIC(HOME_COND_OK_STN1)XIO(RST_SEQ_ON_STN1)XIO(FAULTED_STN1)XIO(CONS_CALB_ON_STN1)MOV(50,MSG_STN1);
   14: XIC(CONSTRICTION_CALB_SEL_STN1)[XIC(START_PB_ONS_STN1) XIC(HOME_COND_OK_STN1) ,XIC(CONS_CALB_ON_STN1) ]XIO(RST_SEQ_ON_STN1)XIO(CONS_CALB_OFF_STN1)OTE(CONS_CALB_ON_STN1);
   15: XIC(CONSTRICTION_CALB_SEL_STN2)XIC(HOME_COND_OK_STN2)XIO(RST_SEQ_ON_STN2)XIO(FAULTED_STN2)XIO(CONS_CALB_ON_STN2)MOV(50,MSG_STN2);
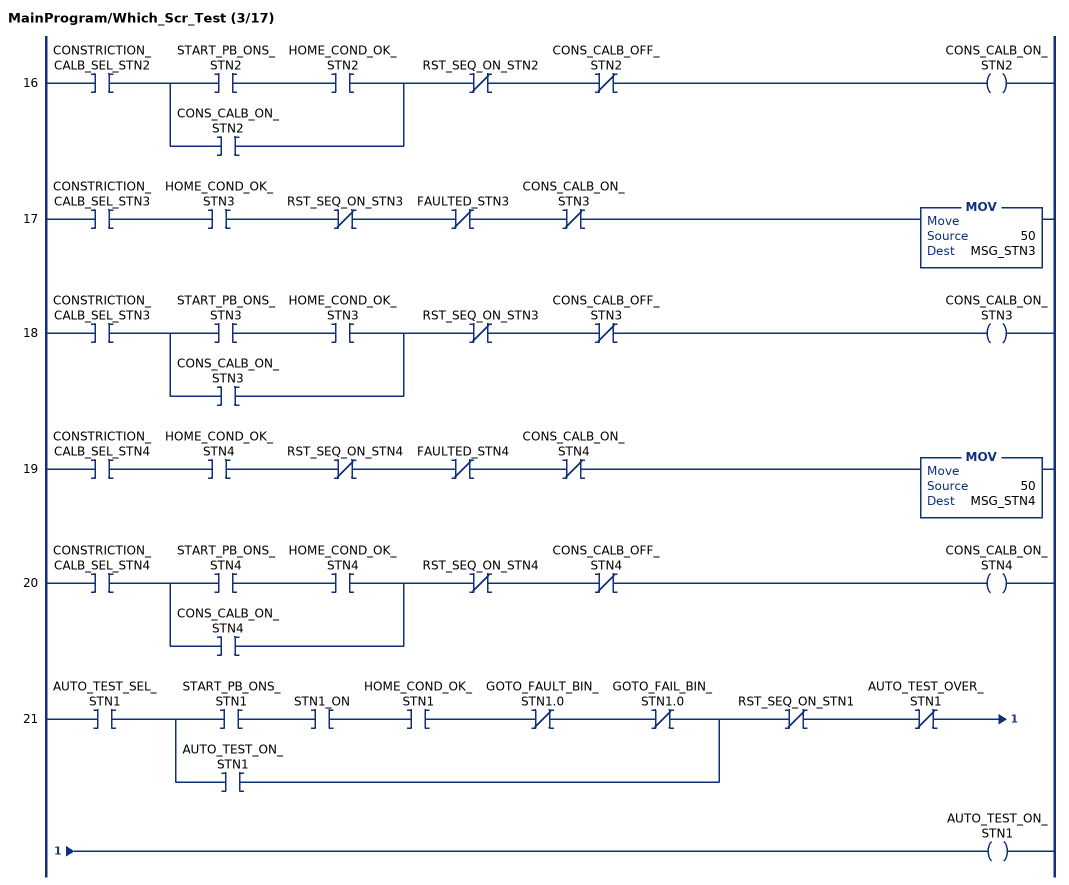
   16: XIC(CONSTRICTION_CALB_SEL_STN2)[XIC(START_PB_ONS_STN2) XIC(HOME_COND_OK_STN2) ,XIC(CONS_CALB_ON_STN2) ]XIO(RST_SEQ_ON_STN2)XIO(CONS_CALB_OFF_STN2)OTE(CONS_CALB_ON_STN2);
   17: XIC(CONSTRICTION_CALB_SEL_STN3)XIC(HOME_COND_OK_STN3)XIO(RST_SEQ_ON_STN3)XIO(FAULTED_STN3)XIO(CONS_CALB_ON_STN3)MOV(50,MSG_STN3);
   18: XIC(CONSTRICTION_CALB_SEL_STN3)[XIC(START_PB_ONS_STN3) XIC(HOME_COND_OK_STN3) ,XIC(CONS_CALB_ON_STN3) ]XIO(RST_SEQ_ON_STN3)XIO(CONS_CALB_OFF_STN3)OTE(CONS_CALB_ON_STN3);
   19: XIC(CONSTRICTION_CALB_SEL_STN4)XIC(HOME_COND_OK_STN4)XIO(RST_SEQ_ON_STN4)XIO(FAULTED_STN4)XIO(CONS_CALB_ON_STN4)MOV(50,MSG_STN4);
   20: XIC(CONSTRICTION_CALB_SEL_STN4)[XIC(START_PB_ONS_STN4) XIC(HOME_COND_OK_STN4) ,XIC(CONS_CALB_ON_STN4) ]XIO(RST_SEQ_ON_STN4)XIO(CONS_CALB_OFF_STN4)OTE(CONS_CALB_ON_STN4);
   21: XIC(AUTO_TEST_SEL_STN1)[XIC(START_PB_ONS_STN1) XIC(STN1_ON) XIC(HOME_COND_OK_STN1) XIO(GOTO_FAULT_BIN_STN1.0) XIO(GOTO_FAIL_BIN_STN1.0) ,XIC(AUTO_TEST_ON_STN1) ]XIO(RST_SEQ_ON_STN1)XIO(AUTO_TEST_OVER_STN1)OTE(AUTO_TEST_ON_STN1);
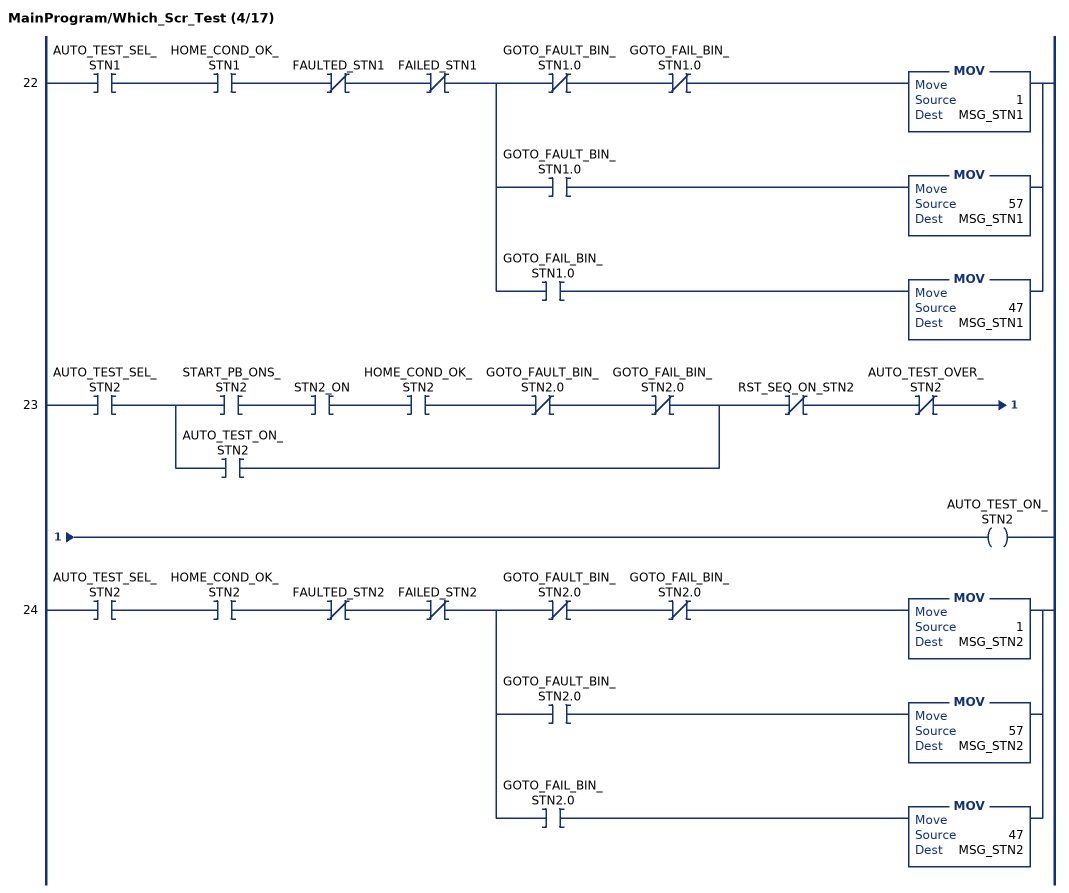
   22: XIC(AUTO_TEST_SEL_STN1)XIC(HOME_COND_OK_STN1)XIO(FAULTED_STN1)XIO(FAILED_STN1)[XIO(GOTO_FAULT_BIN_STN1.0) XIO(GOTO_FAIL_BIN_STN1.0) MOV(1,MSG_STN1) ,XIC(GOTO_FAULT_BIN_STN1.0) MOV(57,MSG_STN1) ,XIC(GOTO_FAIL_BIN_STN1.0) MOV(47,MSG_STN1) ];
   23: XIC(AUTO_TEST_SEL_STN2)[XIC(START_PB_ONS_STN2) XIC(STN2_ON) XIC(HOME_COND_OK_STN2) XIO(GOTO_FAULT_BIN_STN2.0) XIO(GOTO_FAIL_BIN_STN2.0) ,XIC(AUTO_TEST_ON_STN2) ]XIO(RST_SEQ_ON_STN2)XIO(AUTO_TEST_OVER_STN2)OTE(AUTO_TEST_ON_STN2);
   24: XIC(AUTO_TEST_SEL_STN2)XIC(HOME_COND_OK_STN2)XIO(FAULTED_STN2)XIO(FAILED_STN2)[XIO(GOTO_FAULT_BIN_STN2.0) XIO(GOTO_FAIL_BIN_STN2.0) MOV(1,MSG_STN2) ,XIC(GOTO_FAULT_BIN_STN2.0) MOV(57,MSG_STN2) ,XIC(GOTO_FAIL_BIN_STN2.0) MOV(47,MSG_STN2) ];
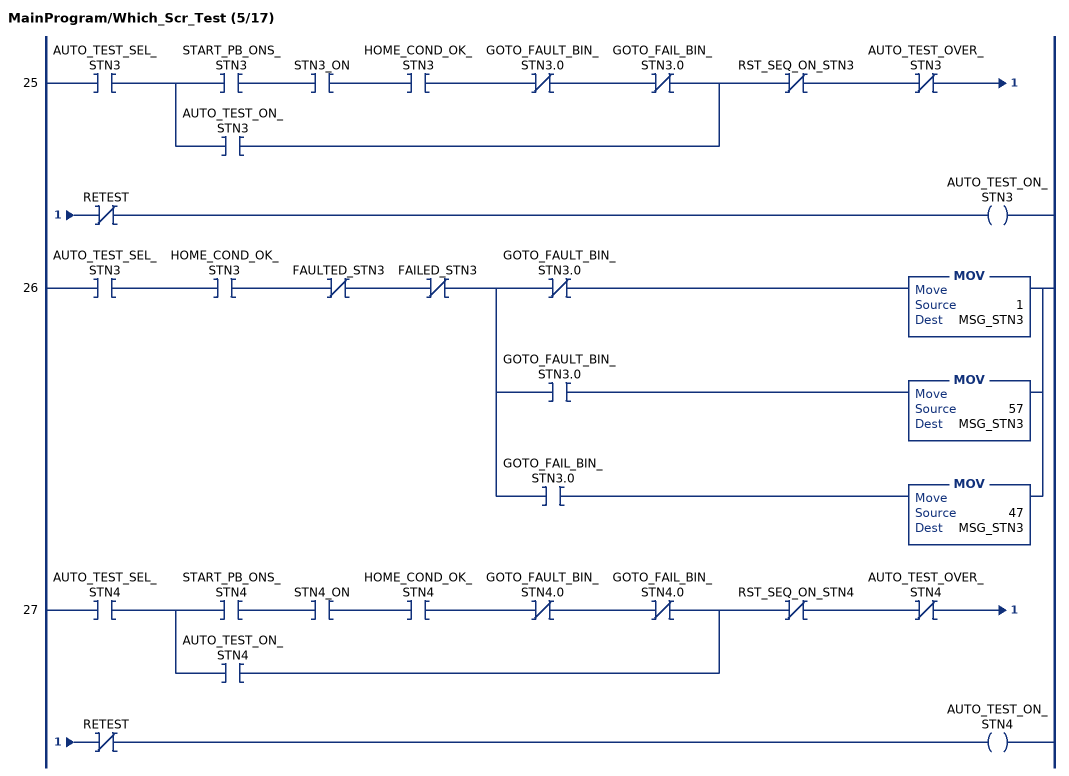
   25: XIC(AUTO_TEST_SEL_STN3)[XIC(START_PB_ONS_STN3) XIC(STN3_ON) XIC(HOME_COND_OK_STN3) XIO(GOTO_FAULT_BIN_STN3.0) XIO(GOTO_FAIL_BIN_STN3.0) ,XIC(AUTO_TEST_ON_STN3) ]XIO(RST_SEQ_ON_STN3)XIO(AUTO_TEST_OVER_STN3)XIO(RETEST)OTE(AUTO_TEST_ON_STN3);
   26: XIC(AUTO_TEST_SEL_STN3)XIC(HOME_COND_OK_STN3)XIO(FAULTED_STN3)XIO(FAILED_STN3)[XIO(GOTO_FAULT_BIN_STN3.0) MOV(1,MSG_STN3) ,XIC(GOTO_FAULT_BIN_STN3.0) MOV(57,MSG_STN3) ,XIC(GOTO_FAIL_BIN_STN3.0) MOV(47,MSG_STN3) ];
   27: XIC(AUTO_TEST_SEL_STN4)[XIC(START_PB_ONS_STN4) XIC(STN4_ON) XIC(HOME_COND_OK_STN4) XIO(GOTO_FAULT_BIN_STN4.0) XIO(GOTO_FAIL_BIN_STN4.0) ,XIC(AUTO_TEST_ON_STN4) ]XIO(RST_SEQ_ON_STN4)XIO(AUTO_TEST_OVER_STN4)XIO(RETEST)OTE(AUTO_TEST_ON_STN4);
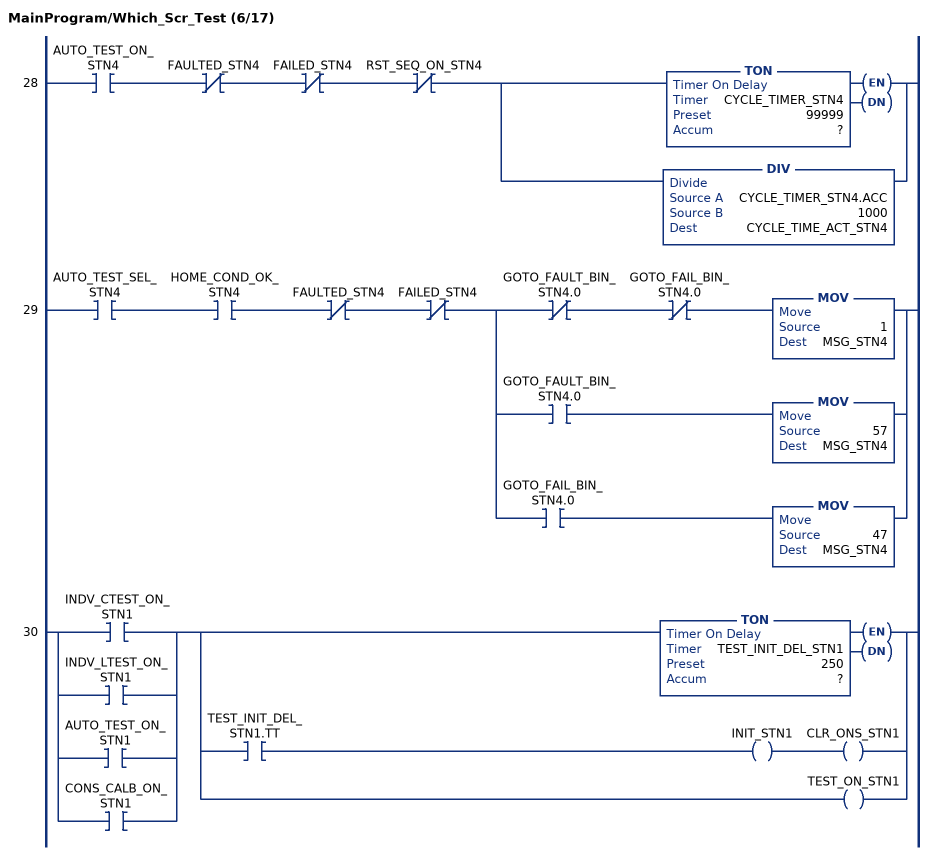
   28: XIC(AUTO_TEST_ON_STN4)XIO(FAULTED_STN4)XIO(FAILED_STN4)XIO(RST_SEQ_ON_STN4)[TON(CYCLE_TIMER_STN4,?,?) ,DIV(CYCLE_TIMER_STN4.ACC,1000,CYCLE_TIME_ACT_STN4) ];
   29: XIC(AUTO_TEST_SEL_STN4)XIC(HOME_COND_OK_STN4)XIO(FAULTED_STN4)XIO(FAILED_STN4)[XIO(GOTO_FAULT_BIN_STN4.0) XIO(GOTO_FAIL_BIN_STN4.0) MOV(1,MSG_STN4) ,XIC(GOTO_FAULT_BIN_STN4.0) MOV(57,MSG_STN4) ,XIC(GOTO_FAIL_BIN_STN4.0) MOV(47,MSG_STN4) ];
   30: [XIC(INDV_CTEST_ON_STN1) ,XIC(INDV_LTEST_ON_STN1) ,XIC(AUTO_TEST_ON_STN1) ,XIC(CONS_CALB_ON_STN1) ][TON(TEST_INIT_DEL_STN1,?,?) ,XIC(TEST_INIT_DEL_STN1.TT) OTE(INIT_STN1) OTE(CLR_ONS_STN1) ,OTE(TEST_ON_STN1) ];
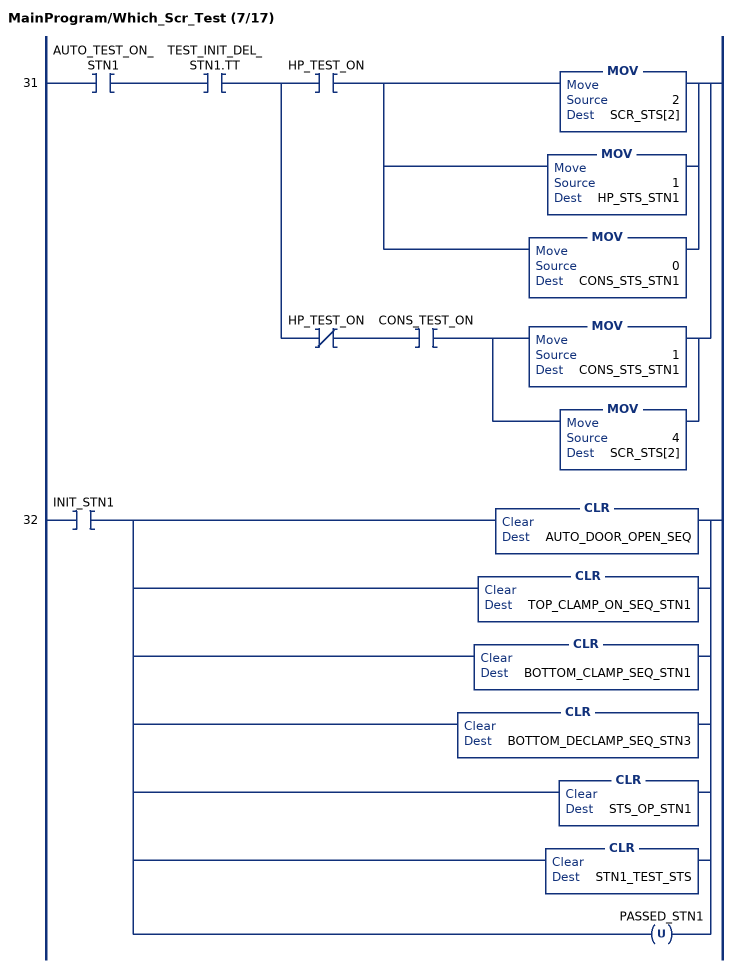
   31: XIC(AUTO_TEST_ON_STN1)XIC(TEST_INIT_DEL_STN1.TT)[XIC(HP_TEST_ON) [MOV(2,SCR_STS[2]) ,MOV(1,HP_STS_STN1) ,MOV(0,CONS_STS_STN1) ] ,XIO(HP_TEST_ON) XIC(CONS_TEST_ON) [MOV(1,CONS_STS_STN1) ,MOV(4,SCR_STS[2]) ] ];
   32: XIC(INIT_STN1)[CLR(AUTO_DOOR_OPEN_SEQ) ,CLR(TOP_CLAMP_ON_SEQ_STN1) ,CLR(BOTTOM_CLAMP_SEQ_STN1) ,CLR(BOTTOM_DECLAMP_SEQ_STN3) ,CLR(STS_OP_STN1) ,CLR(STN1_TEST_STS) ,OTU(PASSED_STN1) ];
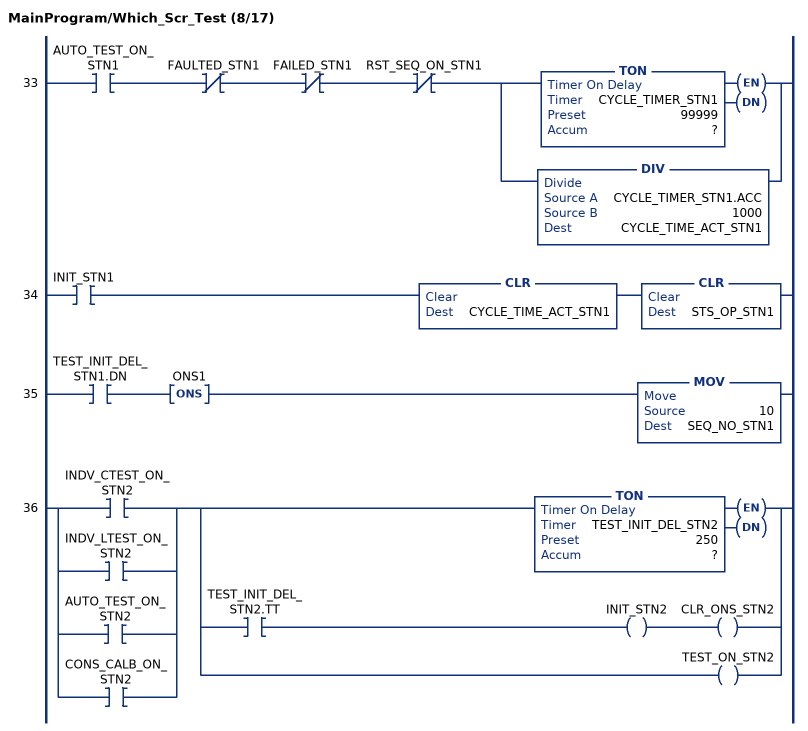
   33: XIC(AUTO_TEST_ON_STN1)XIO(FAULTED_STN1)XIO(FAILED_STN1)XIO(RST_SEQ_ON_STN1)[TON(CYCLE_TIMER_STN1,?,?) ,DIV(CYCLE_TIMER_STN1.ACC,1000,CYCLE_TIME_ACT_STN1) ];
   34: XIC(INIT_STN1)CLR(CYCLE_TIME_ACT_STN1)CLR(STS_OP_STN1);
   35: XIC(TEST_INIT_DEL_STN1.DN)ONS(ONS1)MOV(10,SEQ_NO_STN1);
   36: [XIC(INDV_CTEST_ON_STN2) ,XIC(INDV_LTEST_ON_STN2) ,XIC(AUTO_TEST_ON_STN2) ,XIC(CONS_CALB_ON_STN2) ][TON(TEST_INIT_DEL_STN2,?,?) ,XIC(TEST_INIT_DEL_STN2.TT) OTE(INIT_STN2) OTE(CLR_ONS_STN2) ,OTE(TEST_ON_STN2) ];
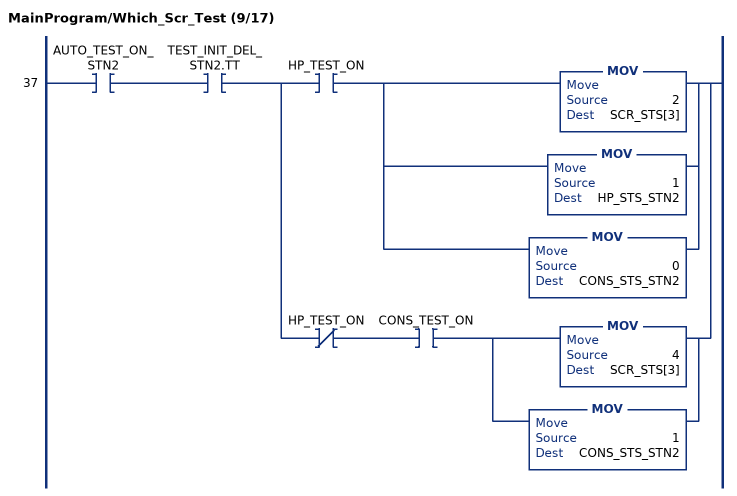
   37: XIC(AUTO_TEST_ON_STN2)XIC(TEST_INIT_DEL_STN2.TT)[XIC(HP_TEST_ON) [MOV(2,SCR_STS[3]) ,MOV(1,HP_STS_STN2) ,MOV(0,CONS_STS_STN2) ] ,XIO(HP_TEST_ON) XIC(CONS_TEST_ON) [MOV(4,SCR_STS[3]) ,MOV(1,CONS_STS_STN2) ] ];
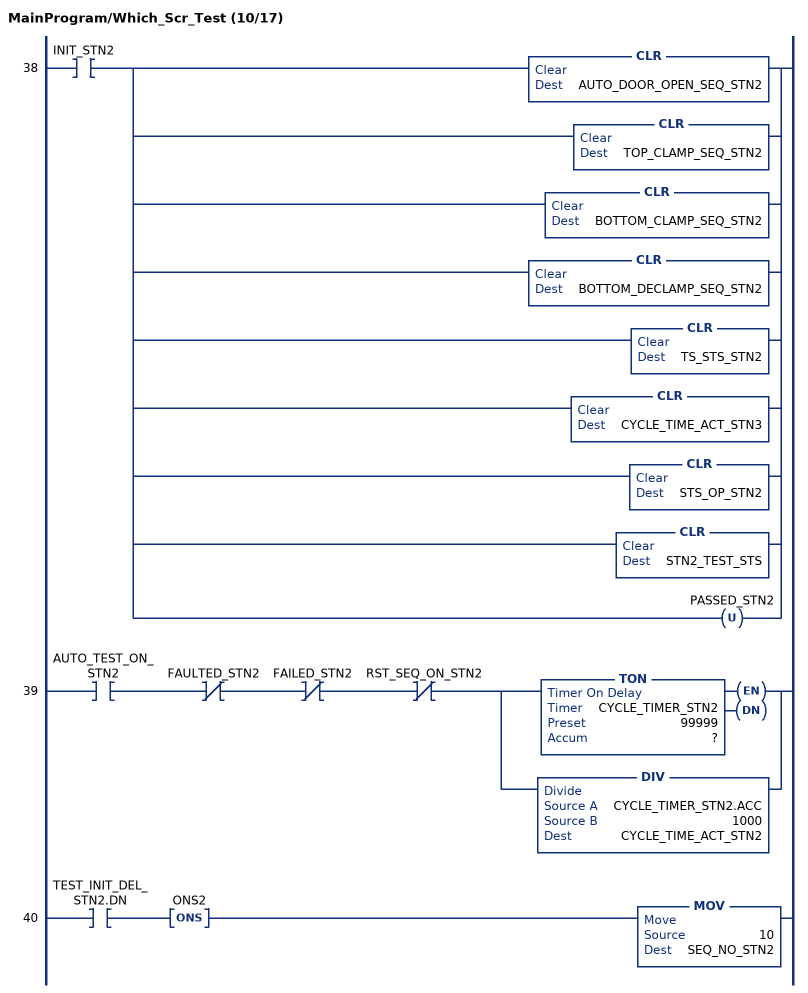
   38: XIC(INIT_STN2)[CLR(AUTO_DOOR_OPEN_SEQ_STN2) ,CLR(TOP_CLAMP_SEQ_STN2) ,CLR(BOTTOM_CLAMP_SEQ_STN2) ,CLR(BOTTOM_DECLAMP_SEQ_STN2) ,CLR(TS_STS_STN2) ,CLR(CYCLE_TIME_ACT_STN3) ,CLR(STS_OP_STN2) ,CLR(STN2_TEST_STS) ,OTU(PASSED_STN2) ];
   39: XIC(AUTO_TEST_ON_STN2)XIO(FAULTED_STN2)XIO(FAILED_STN2)XIO(RST_SEQ_ON_STN2)[TON(CYCLE_TIMER_STN2,?,?) ,DIV(CYCLE_TIMER_STN2.ACC,1000,CYCLE_TIME_ACT_STN2) ];
   40: XIC(TEST_INIT_DEL_STN2.DN)ONS(ONS2)MOV(10,SEQ_NO_STN2);
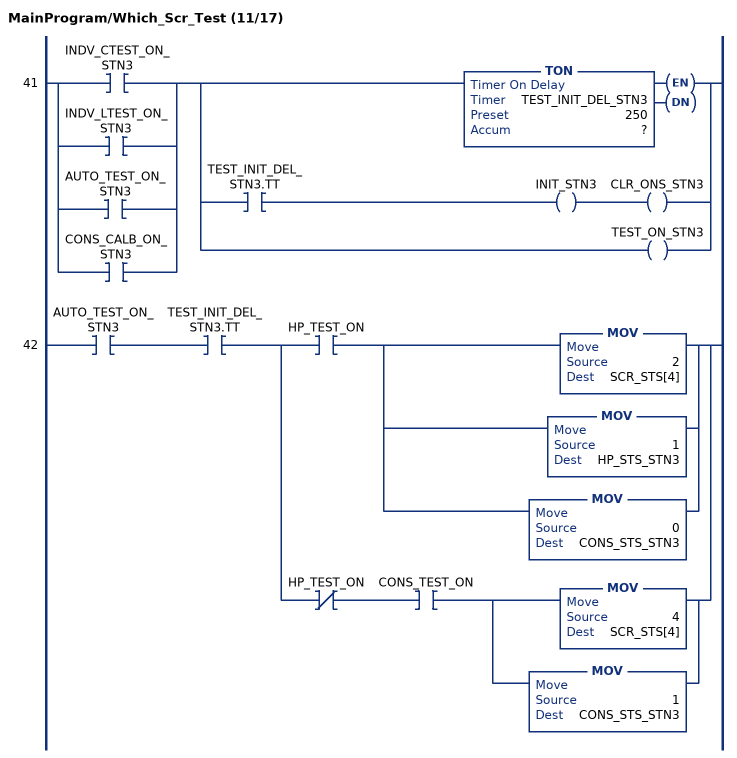
   41: [XIC(INDV_CTEST_ON_STN3) ,XIC(INDV_LTEST_ON_STN3) ,XIC(AUTO_TEST_ON_STN3) ,XIC(CONS_CALB_ON_STN3) ][TON(TEST_INIT_DEL_STN3,?,?) ,XIC(TEST_INIT_DEL_STN3.TT) OTE(INIT_STN3) OTE(CLR_ONS_STN3) ,OTE(TEST_ON_STN3) ];
   42: XIC(AUTO_TEST_ON_STN3)XIC(TEST_INIT_DEL_STN3.TT)[XIC(HP_TEST_ON) [MOV(2,SCR_STS[4]) ,MOV(1,HP_STS_STN3) ,MOV(0,CONS_STS_STN3) ] ,XIO(HP_TEST_ON) XIC(CONS_TEST_ON) [MOV(4,SCR_STS[4]) ,MOV(1,CONS_STS_STN3) ] ];
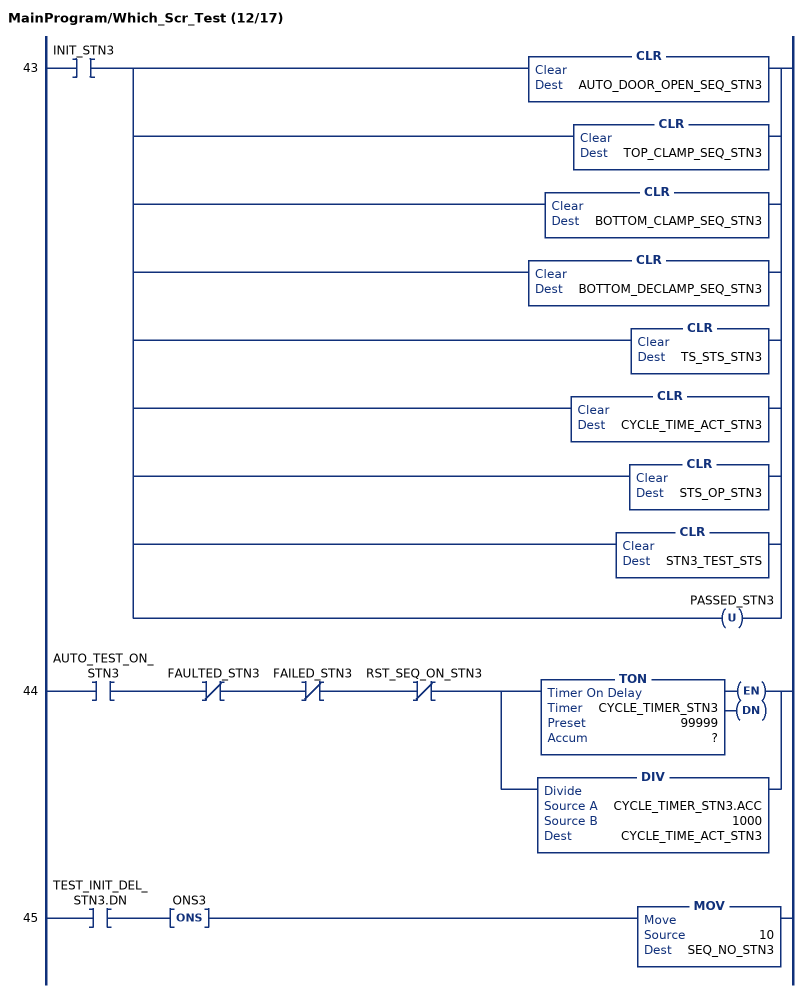
   43: XIC(INIT_STN3)[CLR(AUTO_DOOR_OPEN_SEQ_STN3) ,CLR(TOP_CLAMP_SEQ_STN3) ,CLR(BOTTOM_CLAMP_SEQ_STN3) ,CLR(BOTTOM_DECLAMP_SEQ_STN3) ,CLR(TS_STS_STN3) ,CLR(CYCLE_TIME_ACT_STN3) ,CLR(STS_OP_STN3) ,CLR(STN3_TEST_STS) ,OTU(PASSED_STN3) ];
   44: XIC(AUTO_TEST_ON_STN3)XIO(FAULTED_STN3)XIO(FAILED_STN3)XIO(RST_SEQ_ON_STN3)[TON(CYCLE_TIMER_STN3,?,?) ,DIV(CYCLE_TIMER_STN3.ACC,1000,CYCLE_TIME_ACT_STN3) ];
   45: XIC(TEST_INIT_DEL_STN3.DN)ONS(ONS3)MOV(10,SEQ_NO_STN3);
